Yaskawa INFORM job: X2_48(150,-90).JBI

/JOB
//NAME X2_48(150,-90)
//POS
///NPOS 102,102,102,5,0,0
///TOOL 0
///POSTYPE PULSE
///PULSE
C00000=2000,-112988,-119327,0,83158,0
C00001=-142756,-112988,-119327,-18089,83158,34222
C00002=-145489,-137180,-128771,-21394,87700,32111
C00003=-164591,-94889,-79086,-18920,74682,27376
C00004=-167906,-89992,-74155,-18360,73432,26351
C00005=-169175,-88015,-72150,-18139,72941,25959
C00006=-169090,-86796,-69106,-18271,71772,26171
C00007=-169175,-88015,-72150,-18139,72941,25959
C00008=-170099,-88727,-72164,-17993,72396,25701
C00009=-172764,-85592,-70856,-17391,72586,24688
C00010=-170099,-88727,-72164,-17993,72396,25701
C00011=-185420,-95958,-68594,7326,50076,11474
C00012=-182716,-92695,-67464,5857,50831,12695
C00013=-185420,-95958,-68594,7326,50076,11474
C00014=-184506,-107402,-76413,6968,48935,11790
C00015=-159220,-109944,-102922,-24512,66979,45642
C00016=-167824,-173568,-124205,-26542,46564,47026
C00017=-170252,-85554,-47492,-36176,17718,77515
C00018=-172784,-79149,-41877,-32040,16598,75352
C00019=-173728,-76594,-39584,-30409,16175,74507
C00020=-175520,-74869,-38841,-26085,15969,72339
C00021=-173728,-76594,-39584,-30409,16175,74507
C00022=-175036,-75380,-39094,-27253,16023,72924
C00023=-174520,-73484,-36544,-29303,15665,73921
C00024=-175036,-75380,-39094,-27253,16023,72924
C00025=-171703,-84374,-47061,-33102,17430,75946
C00026=-118222,-104921,-85597,2302,76232,-3756
C00027=-70971,-85923,-48405,35291,17571,-76879
C00028=-68458,-79485,-42811,31017,16504,-74660
C00029=-67521,-76918,-40527,29335,16103,-73795
C00030=-65747,-75173,-39789,24982,15938,-71620
C00031=-67521,-76918,-40527,29335,16103,-73795
C00032=-66355,-75782,-40029,26507,15971,-72380
C00033=-66862,-73889,-37487,28530,15606,-73362
C00034=-66355,-75782,-40029,26507,15971,-72380
C00035=-67257,-78357,-42329,28198,16341,-73244
C00036=-69676,-84817,-47961,32519,17317,-75468
C00037=-66595,-165951,-119904,20395,34837,-49941
C00038=-38828,-178555,-122254,-18105,43219,-2401
C00039=-76877,-95412,-79683,19208,74450,-27234
C00040=-73543,-90451,-74757,18629,73220,-26200
C00041=-72268,-88450,-72755,18400,72736,-25804
C00042=-72333,-87219,-69709,18531,71571,-26012
C00043=-72268,-88450,-72755,18400,72736,-25804
C00044=-71656,-87743,-71624,18310,72282,-25648
C00045=-69017,-84617,-70326,17702,72469,-24642
C00046=-71656,-87743,-71624,18310,72282,-25648
C00047=-55558,-95793,-69122,-7502,50260,-11083
C00048=-58281,-92556,-67996,-6016,50996,-12311
C00049=-55558,-95793,-69122,-7502,50260,-11083
C00050=-56403,-107290,-76939,-7182,49095,-11365
C00051=-66823,-91712,-74133,7065,60566,-19717
C00052=-66824,-90415,-70771,7163,59174,-19807
C00053=-66824,-89866,-69409,7204,58621,-19844
C00054=-66826,-90728,-71569,20336,73429,-25465
C00055=-66823,-90174,-70167,23017,76716,-26688
C00056=-65098,-92992,-71165,22907,75465,-26287
C00057=-62596,-96858,-72515,22741,73703,-25691
C00058=-66824,-90716,-71530,22972,77234,-26586
C00059=-66823,-92043,-75030,22863,78594,-26321
C00060=-119458,-64652,-78063,7993,91912,-2412
C00061=-162081,-130804,-92299,-12648,53591,25594
C00062=-176554,-94726,-71925,-6352,57827,19319
C00063=-177319,-91851,-69580,-6047,57801,19017
C00064=-164142,-69988,-61942,-21167,80883,28211
C00065=-180907,-101373,-74314,-19437,68720,24090
C00066=-178862,-97024,-72377,-22464,73935,25818
C00067=-182257,-101563,-73927,-22219,71739,24962
C00068=-185323,-105109,-74952,-21976,69813,24167
C00069=-177337,-98931,-74291,-22610,74536,26275
C00070=-148639,-128504,-104999,-23996,86118,34643
C00071=-125763,-70435,-126192,3026,94587,-28672
C00072=-71267,-74397,-112769,-20427,89435,-13482
C00073=-68499,-138788,-124688,10863,39680,-60380
C00074=-66279,-93192,-102590,7723,49796,-58218
C00075=-66723,-80903,-95652,7638,51727,-58168
C00076=-67166,-79691,-95913,8650,53907,-57954
C00077=-66992,-84383,-98076,16350,53747,-64312
C00078=-66975,-84373,-97955,15118,51249,-65099
C00079=-67019,-84412,-97997,13413,47585,-66286
C00080=-67040,-84369,-98104,11818,43956,-67447
C00081=-67158,-84518,-98164,9623,37605,-69507
C00082=-63016,-95130,-103823,1707,27635,-69538
C00083=-60476,-99306,-104126,-2746,25300,-67760
C00084=-58396,-103594,-105732,-6580,24205,-66047
C00085=-71788,-113583,-131480,12468,38511,-72889
C00086=-126548,-133354,-124162,3479,55623,-10129
C00087=-185990,-110059,-108050,-2198,41333,59059
C00088=-176703,-90185,-100504,-9996,47566,62974
C00089=-174384,-84529,-98133,-11690,49287,63786
C00090=-173672,-80861,-96753,-12075,50409,63954
C00091=-174317,-84499,-98582,-11694,49583,63780
C00092=-175157,-86850,-99377,-16101,54637,63302
C00093=-174420,-84357,-98340,-15790,53093,64898
C00094=-174441,-84329,-98230,-14052,49361,66088
C00095=-174408,-84392,-98156,-13024,46821,66903
C00096=-174442,-84322,-97937,-10190,39158,69319
C00097=-177828,-93138,-101730,-4745,30921,69477
C00098=-180987,-99716,-104277,2046,25458,68211
C00099=-183030,-103926,-105848,5755,24360,66553
C00100=-165604,-146579,-119354,-35431,57728,66075
C00101=2000,-112988,-119327,0,83158,0
BC00000=91901,666204,1075175
BC00001=176532,676723,1075175
BC00002=176532,817677,1075175
BC00003=176532,817677,1075175
BC00004=176532,817677,1075175
BC00005=176532,817677,1075175
BC00006=176532,817677,1075175
BC00007=176532,817677,1075175
BC00008=176532,817677,1075175
BC00009=176532,817677,1075175
BC00010=176532,817677,1075175
BC00011=176532,817677,1075175
BC00012=176532,817677,1075175
BC00013=176532,817677,1075175
BC00014=176532,817677,1075175
BC00015=185949,779707,1075175
BC00016=185949,764059,1075175
BC00017=201887,715451,1075175
BC00018=201887,715451,1075175
BC00019=201887,715451,1075175
BC00020=201887,715451,1075175
BC00021=201887,715451,1075175
BC00022=201887,715451,1075175
BC00023=201887,715451,1075175
BC00024=201887,715451,1075175
BC00025=201887,715451,1075175
BC00026=220159,715941,1075175
BC00027=236281,716374,1075175
BC00028=236281,716374,1075175
BC00029=236281,716374,1075175
BC00030=236281,716374,1075175
BC00031=236281,716374,1075175
BC00032=236281,716374,1075175
BC00033=236281,716374,1075175
BC00034=236281,716374,1075175
BC00035=236281,716374,1075175
BC00036=221001,696814,1073215
BC00037=243248,739230,1070806
BC00038=260118,819465,1075175
BC00039=260118,819465,1075175
BC00040=260118,819465,1075175
BC00041=260118,819465,1075175
BC00042=260118,819465,1075175
BC00043=260118,819465,1075175
BC00044=260118,819465,1075175
BC00045=260118,819465,1075175
BC00046=260118,819465,1075175
BC00047=260118,819465,1075175
BC00048=260118,819465,1075175
BC00049=260118,819465,1075175
BC00050=260118,819465,1075175
BC00051=256603,821231,1075175
BC00052=262054,823449,1075175
BC00053=264234,824336,1075175
BC00054=261899,852526,1075175
BC00055=262928,818909,1075175
BC00056=262928,818909,1075175
BC00057=262928,818909,1075175
BC00058=260700,819348,1075175
BC00059=255130,820445,1075175
BC00060=215695,750105,1075175
BC00061=173796,826500,1075175
BC00062=173796,826500,1075175
BC00063=173796,826500,1075175
BC00064=173796,826500,1075175
BC00065=173796,826500,1075175
BC00066=173796,826500,1075175
BC00067=173796,826500,1075175
BC00068=173796,826500,1075175
BC00069=173796,826500,1075175
BC00070=173796,826500,1075175
BC00071=206784,690000,907696
BC00072=206784,667756,907696
BC00073=237138,734038,765099
BC00074=234870,735507,776012
BC00075=235241,735609,774811
BC00076=235241,735609,774812
BC00077=230700,738342,767293
BC00078=230768,725722,749509
BC00079=230851,711605,722921
BC00080=230958,694408,685041
BC00081=231101,675536,626400
BC00082=231249,666513,542099
BC00083=229011,666220,543730
BC00084=223399,666220,557733
BC00085=223385,666220,578143
BC00086=226917,670779,831730
BC00087=230837,715030,776411
BC00088=213006,734477,776411
BC00089=207409,735992,758036
BC00090=206083,736350,753680
BC00091=205170,736598,750685
BC00092=206638,744474,770770
BC00093=207359,723163,745950
BC00094=207429,712052,723300
BC00095=207513,698239,694954
BC00096=207680,674502,624413
BC00097=207794,669496,570286
BC00098=210112,666220,540525
BC00099=215722,666220,554666
BC00100=215722,666220,928985
BC00101=91901,666204,1075175
EC00000=1330261,-556475
EC00001=1330261,-556475
EC00002=1330261,-556475
EC00003=1330261,-556475
EC00004=1330261,-556475
EC00005=1330261,-556475
EC00006=1330261,-556475
EC00007=1330261,-556475
EC00008=1330261,-556475
EC00009=1330261,-556475
EC00010=1330261,-556475
EC00011=1330261,-556475
EC00012=1330261,-556475
EC00013=1330261,-556475
EC00014=1330261,-556475
EC00015=1330261,-556475
EC00016=1330261,-556475
EC00017=1330261,-556475
EC00018=1330261,-556475
EC00019=1330261,-556475
EC00020=1330261,-556475
EC00021=1330261,-556475
EC00022=1330261,-556475
EC00023=1330261,-556475
EC00024=1330261,-556475
EC00025=1330261,-556475
EC00026=1330261,-556475
EC00027=1330261,-556475
EC00028=1330261,-556475
EC00029=1330261,-556475
EC00030=1330261,-556475
EC00031=1330261,-556475
EC00032=1330261,-556475
EC00033=1330261,-556475
EC00034=1330261,-556475
EC00035=1330261,-556475
EC00036=1330261,-556475
EC00037=1330261,-556475
EC00038=1330261,-556475
EC00039=1330261,-556475
EC00040=1330261,-556475
EC00041=1330261,-556475
EC00042=1330261,-556475
EC00043=1330261,-556475
EC00044=1330261,-556475
EC00045=1330261,-556475
EC00046=1330261,-556475
EC00047=1330261,-556475
EC00048=1330261,-556475
EC00049=1330261,-556475
EC00050=1330261,-556475
EC00051=1330261,-556475
EC00052=1330261,-556475
EC00053=1330261,-556475
EC00054=1330261,-556475
EC00055=1330261,-556475
EC00056=1330261,-556475
EC00057=1330261,-556475
EC00058=1330261,-556475
EC00059=1330261,-556475
EC00060=1330261,-556475
EC00061=1330261,-556475
EC00062=1330261,-556475
EC00063=1330261,-556475
EC00064=1330261,-556475
EC00065=1330261,-556475
EC00066=1330261,-556475
EC00067=1330261,-556475
EC00068=1330261,-556475
EC00069=1330261,-556475
EC00070=1330261,-556475
EC00071=1330261,-556475
EC00072=1330261,-556475
EC00073=1330261,-556475
EC00074=1330261,-556475
EC00075=1330261,-556474
EC00076=1330261,-556475
EC00077=1330261,-556475
EC00078=1330261,-556475
EC00079=1330261,-556475
EC00080=1330261,-556475
EC00081=1330261,-556475
EC00082=1330261,-556475
EC00083=1330261,-556475
EC00084=1330261,-556475
EC00085=1330261,-556475
EC00086=1330261,-556475
EC00087=1330261,-556475
EC00088=1330261,-556475
EC00089=1330261,-556475
EC00090=1330261,-556474
EC00091=1330261,-556475
EC00092=1330261,-556475
EC00093=1330261,-556475
EC00094=1330261,-556475
EC00095=1330261,-556475
EC00096=1330261,-556475
EC00097=1330261,-556475
EC00098=1330261,-556475
EC00099=1330261,-556475
EC00100=1330261,-556475
EC00101=1330261,-556475
///POSTYPE BASE
///RECTAN
///RCONF 0,0,0,0,0,0,0,0,0,0,0,0,0,0,0,0,0,0,0,0,0,0,0,0
P00006=9.046,-3.472,-3.145,0.0000,0.0000,0.0000
P00021=3.198,-0.012,-3.236,0.0000,0.0000,0.0000
P00022=7.754,0.769,-4.150,0.0000,0.0000,0.0000
P00031=1.853,-0.001,-1.549,0.0000,0.0000,0.0000
P00032=1.957,0.503,-7.217,0.0000,0.0000,0.0000
//INST
///DATE 2025/03/25 13:08
///ATTR SC,RW
///GROUP1 RB1,BS1
///GROUP2 ST1
NOP
'X2_48(150,-90)
MOVJ C00000 BC00000 VJ=100.00  +MOVJ EC00000 VJ=100.00
MOVJ C00001 BC00001 VJ=100.00  +MOVJ EC00001 VJ=100.00
MOVJ C00002 BC00002 VJ=100.00  +MOVJ EC00002 VJ=100.00
'Path S3695
SFTOF3D
MOVJ C00003 BC00003 VJ=100.00  +MOVJ EC00003 VJ=100.00
MOVL C00004 BC00004 V=800.0  +MOVJ EC00004 VJ=100.00
SMOVL C00005 BC00005 V=166.7  +MOVJ EC00005
SREFP 3 C00006 BC00006  +REFP EC00006
CALL JOB:SEARCH-R1-S13D
SET P032 P006
SFTON3D P032
SMOVL C00007 BC00007 V=166.7  +MOVJ EC00007
SMOVL C00008 BC00008 V=166.7  +MOVJ EC00008
SREFP 3 C00009 BC00009  +REFP EC00009
CALL JOB:SEARCH-R1-S13D
SET P032 P006
SFTON3D P032
SMOVL C00010 BC00010 V=166.7  +MOVJ EC00010
SMOVL C00011 BC00011 V=166.7  +MOVJ EC00011
SREFP 3 C00012 BC00012  +REFP EC00012
CALL JOB:SEARCH-R1-S13D
SET P032 P006
SFTON3D P032
SMOVL C00013 BC00013 V=166.7  +MOVJ EC00013
MOVL C00014 BC00014 V=1000.0  +MOVJ EC00014 VJ=100.00
'EndPath S3695
MOVJ C00015 BC00015 VJ=100.00  +MOVJ EC00015 VJ=100.00
MOVJ C00016 BC00016 VJ=100.00  +MOVJ EC00016 VJ=100.00
'Path S3694
SFTOF3D
MOVJ C00017 BC00017 VJ=100.00  +MOVJ EC00017 VJ=100.00
MOVL C00018 BC00018 V=800.0  +MOVJ EC00018 VJ=100.00
SMOVL C00019 BC00019 V=166.7  +MOVJ EC00019
SREFP 3 C00020 BC00020  +REFP EC00020
CALL JOB:SEARCH-R1-S13D
SET P022 P006
SFTON3D P022
SMOVL C00021 BC00021 V=166.7  +MOVJ EC00021
SMOVL C00022 BC00022 V=166.7  +MOVJ EC00022
SREFP 3 C00023 BC00023  +REFP EC00023
CALL JOB:SEARCH-R1-S13D
SET P022 P006
SFTON3D P022
SMOVL C00024 BC00024 V=166.7  +MOVJ EC00024
MOVL C00025 BC00025 V=1000.0  +MOVJ EC00025 VJ=100.00
'EndPath S3694
MOVJ C00026 BC00026 VJ=100.00  +MOVJ EC00026 VJ=100.00
'Path S3696
SFTOF3D
MOVJ C00027 BC00027 VJ=100.00  +MOVJ EC00027 VJ=100.00
MOVL C00028 BC00028 V=800.0  +MOVJ EC00028 VJ=100.00
SMOVL C00029 BC00029 V=166.7  +MOVJ EC00029
SREFP 3 C00030 BC00030  +REFP EC00030
CALL JOB:SEARCH-R1-S13D
SET P021 P006
SFTON3D P021
SMOVL C00031 BC00031 V=166.7  +MOVJ EC00031
SMOVL C00032 BC00032 V=166.7  +MOVJ EC00032
SREFP 3 C00033 BC00033  +REFP EC00033
CALL JOB:SEARCH-R1-S13D
SET P021 P006
SFTON3D P021
SMOVL C00034 BC00034 V=166.7  +MOVJ EC00034
MOVL C00035 BC00035 V=800.0  +MOVJ EC00035 VJ=100.00
MOVL C00036 BC00036 V=1000.0  +MOVJ EC00036 VJ=100.00
'EndPath S3696
MOVJ C00037 BC00037 VJ=100.00  +MOVJ EC00037 VJ=100.00
MOVJ C00038 BC00038 VJ=100.00  +MOVJ EC00038 VJ=100.00
'Path S3697
SFTOF3D
MOVJ C00039 BC00039 VJ=100.00  +MOVJ EC00039 VJ=100.00
MOVL C00040 BC00040 V=800.0  +MOVJ EC00040 VJ=100.00
SMOVL C00041 BC00041 V=166.7  +MOVJ EC00041
SREFP 3 C00042 BC00042  +REFP EC00042
CALL JOB:SEARCH-R1-S13D
SET P031 P006
SFTON3D P031
SMOVL C00043 BC00043 V=166.7  +MOVJ EC00043
SMOVL C00044 BC00044 V=166.7  +MOVJ EC00044
SREFP 3 C00045 BC00045  +REFP EC00045
CALL JOB:SEARCH-R1-S13D
SET P031 P006
SFTON3D P031
SMOVL C00046 BC00046 V=166.7  +MOVJ EC00046
SMOVL C00047 BC00047 V=166.7  +MOVJ EC00047
SREFP 3 C00048 BC00048  +REFP EC00048
CALL JOB:SEARCH-R1-S13D
SET P031 P006
SFTON3D P031
SMOVL C00049 BC00049 V=166.7  +MOVJ EC00049
MOVL C00050 BC00050 V=1000.0  +MOVJ EC00050 VJ=100.00
'EndPath S3697
'Path W3698
SFTOF3D
SFTON3D P031
MOVJ C00051 BC00051 VJ=100.00  +MOVJ EC00051 VJ=100.00
SMOVL C00052 BC00052 V=800.0  +MOVJ EC00052
SMOVL C00053 BC00053 V=166.7 PL=0  +MOVJ EC00053
MACRO1 MJ#(0) ARGF22
ARCON
SMOVL C00054 BC00054 V=10.0  +MOVJ EC00054
SMOVL C00055 BC00055 V=10.0  +MOVJ EC00055
SMOVL C00056 BC00056 V=10.0  +MOVJ EC00056
SMOVL C00057 BC00057 V=10.0  +MOVJ EC00057
ARCOF
SMOVL C00058 BC00058 V=800.0  +MOVJ EC00058
SMOVL C00059 BC00059 V=1000.0  +MOVJ EC00059
SFTOF3D
'EndPath W3698
MOVJ C00060 BC00060 VJ=100.00  +MOVJ EC00060 VJ=100.00
'Path W3699
SFTOF3D
SFTON3D P032
MOVJ C00061 BC00061 VJ=100.00  +MOVJ EC00061 VJ=100.00
SMOVL C00062 BC00062 V=800.0  +MOVJ EC00062
SMOVL C00063 BC00063 V=166.7 PL=0  +MOVJ EC00063
ARCON
SMOVL C00064 BC00064 V=10.0  +MOVJ EC00064
SMOVL C00065 BC00065 V=10.0  +MOVJ EC00065
SMOVL C00066 BC00066 V=10.0  +MOVJ EC00066
SMOVL C00067 BC00067 V=10.0  +MOVJ EC00067
SMOVL C00068 BC00068 V=10.0  +MOVJ EC00068
ARCOF
SMOVL C00069 BC00069 V=800.0  +MOVJ EC00069
MOVJ C00070 BC00070 VJ=100.00  +MOVJ EC00070 VJ=100.00
SFTOF3D
'EndPath W3699
MOVJ C00071 BC00071 VJ=100.00  +MOVJ EC00071 VJ=100.00
MOVJ C00072 BC00072 VJ=100.00  +MOVJ EC00072 VJ=100.00
MOVJ C00073 BC00073 VJ=100.00  +MOVJ EC00073 VJ=100.00
'Path W3700
SFTOF3D
SFTON3D P021
SMOVL C00074 BC00074 V=800.0  +MOVJ EC00074
SMOVL C00075 BC00075 V=333.3  +MOVJ EC00075
ARCON
SMOVC C00076 BC00076 V=10.0  +MOVJ EC00076
SMOVC C00077 BC00077 V=10.0  +MOVJ EC00077
SMOVC C00078 BC00078 V=10.0  +MOVJ EC00078
SMOVC C00079 BC00079 V=10.0  +MOVJ EC00079
SMOVC C00080 BC00080 V=10.0  +MOVJ EC00080
SMOVC C00081 BC00081 V=10.0  +MOVJ EC00081
SMOVC C00082 BC00082 V=10.0  +MOVJ EC00082
ARCOF
SMOVL C00083 BC00083 V=800.0  +MOVJ EC00083
SMOVL C00084 BC00084 V=1000.0  +MOVJ EC00084
SFTOF3D
'EndPath W3700
MOVJ C00085 BC00085 VJ=100.00  +MOVJ EC00085 VJ=100.00
MOVJ C00086 BC00086 VJ=100.00  +MOVJ EC00086 VJ=100.00
MOVJ C00087 BC00087 VJ=100.00  +MOVJ EC00087 VJ=100.00
'Path W4285
SFTOF3D
SFTON3D P022
MOVJ C00088 BC00088 VJ=100.00  +MOVJ EC00088 VJ=100.00
SMOVL C00089 BC00089 V=800.0  +MOVJ EC00089
SMOVC C00090 BC00090 V=150.0 PL=0  +MOVJ EC00090
ARCON
SMOVC C00091 BC00091 V=10.0  +MOVJ EC00091
SMOVC C00092 BC00092 V=10.0  +MOVJ EC00092
SMOVC C00093 BC00093 V=10.0  +MOVJ EC00093
SMOVC C00094 BC00094 V=10.0  +MOVJ EC00094
SMOVC C00095 BC00095 V=10.0  +MOVJ EC00095
SMOVC C00096 BC00096 V=10.0  +MOVJ EC00096
SMOVL C00097 BC00097 V=10.0  +MOVJ EC00097
ARCOF
SMOVL C00098 BC00098 V=800.0  +MOVJ EC00098
SMOVL C00099 BC00099 V=1000.0  +MOVJ EC00099
SFTOF3D
'EndPath W4285
MOVJ C00100 BC00100 VJ=100.00  +MOVJ EC00100 VJ=100.00
MOVJ C00101 BC00101 VJ=100.00  +MOVJ EC00101 VJ=100.00
END
